// TIA Portal project "WASHING MACHIN" (V15)

(* hardware
DEVICE "S7-1200 station_1"  S7-1200 Station
   slot 0: "Rack_0"  S7-1200 Rack  Rack  V1.0
   slot 1: "PLC_1"  CPU 1212C DC/DC/DC  6ES7 212-1AE40-0XB0  V4.2
*)

// ===== PLC "PLC_1"  CPU 1212C DC/DC/DC =====

VAR_GLOBAL   // PLC tag table "Default tag table"
   "PB" AT %M0.1 : Bool;
   "A" AT %M0.2 : Bool;
   "ip" AT %Q0.1 : Bool;
   "F water" AT %Q0.2 : Bool;
   "agitation" AT %Q0.3 : Bool;
   "draining" AT %Q0.4 : Bool;
   "spinning" AT %Q0.5 : Bool;
   "alaram" AT %Q0.6 : Bool;
END_VAR

// folder: System blocks/Program resources

DATA_BLOCK "IEC_Timer_0_DB"   // DB1
{ S7_Optimized_Access := 'TRUE' }
AUTHOR : Simatic
FAMILY : IEC
NAME : IEC_TMR
VERSION : 1.0
// stored: InstanceOfName IEC_TIMER
"IEC_TIMER"
BEGIN
END_DATA_BLOCK

DATA_BLOCK "IEC_Timer_0_DB_1"   // DB2
{ S7_Optimized_Access := 'TRUE' }
AUTHOR : Simatic
FAMILY : IEC
NAME : IEC_TMR
VERSION : 1.0
// stored: InstanceOfName IEC_TIMER
"IEC_TIMER"
BEGIN
END_DATA_BLOCK

DATA_BLOCK "IEC_Timer_0_DB_2"   // DB3
{ S7_Optimized_Access := 'TRUE' }
AUTHOR : Simatic
FAMILY : IEC
NAME : IEC_TMR
VERSION : 1.0
// stored: InstanceOfName IEC_TIMER
"IEC_TIMER"
BEGIN
END_DATA_BLOCK

DATA_BLOCK "IEC_Timer_0_DB_3"   // DB4
{ S7_Optimized_Access := 'TRUE' }
AUTHOR : Simatic
FAMILY : IEC
NAME : IEC_TMR
VERSION : 1.0
// stored: InstanceOfName IEC_TIMER
"IEC_TIMER"
BEGIN
END_DATA_BLOCK

DATA_BLOCK "IEC_Timer_0_DB_4"   // DB5
{ S7_Optimized_Access := 'TRUE' }
AUTHOR : Simatic
FAMILY : IEC
NAME : IEC_TMR
VERSION : 1.0
// stored: InstanceOfName IEC_TIMER
"IEC_TIMER"
BEGIN
END_DATA_BLOCK

// folder: (top level)

ORGANIZATION_BLOCK "Main"   // OB1, LAD, ProgramCycle
TITLE = "Main Program Sweep (Cycle)"
{ S7_Optimized_Access := 'TRUE' }
VERSION : 0.1
   VAR_INPUT
      Initial_Call : Bool;   // Initial call of this OB
      Remanence : Bool;   // =True, if remanent data are available
   END_VAR
   VAR_TEMP   // added for the SCL form of the ladder/FBD networks
      _w1 : Bool;
      _w2 : Bool;
      _w3 : Bool;
      _w4 : Bool;
   END_VAR
BEGIN

REGION Network 1
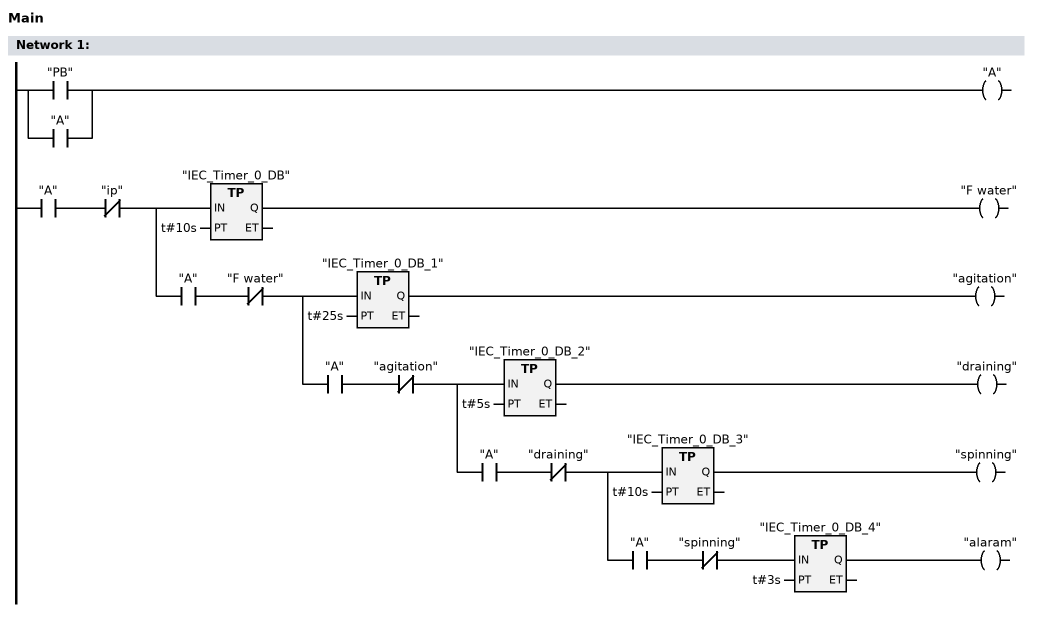
   "A" := "PB" OR "A";
   #_w1 := "A" AND NOT "ip";
   "IEC_Timer_0_DB".TP(IN := #_w1, PT := t#10s);
   "F water" := "IEC_Timer_0_DB".Q;
   #_w2 := #_w1 AND "A" AND NOT "F water";
   "IEC_Timer_0_DB_1".TP(IN := #_w2, PT := t#25s);
   "agitation" := "IEC_Timer_0_DB_1".Q;
   #_w3 := #_w2 AND "A" AND NOT "agitation";
   "IEC_Timer_0_DB_2".TP(IN := #_w3, PT := t#5s);
   "draining" := "IEC_Timer_0_DB_2".Q;
   #_w4 := #_w3 AND "A" AND NOT "draining";
   "IEC_Timer_0_DB_3".TP(IN := #_w4, PT := t#10s);
   "spinning" := "IEC_Timer_0_DB_3".Q;
   "IEC_Timer_0_DB_4".TP(IN := #_w4 AND "A" AND NOT "spinning", PT := t#3s);
   "alaram" := "IEC_Timer_0_DB_4".Q;
END_REGION
END_ORGANIZATION_BLOCK